// TIA Portal V16 export
// export: Created 2022-01-12T14:34:28.4377985Z, ExportSetting WithDefaults, DisplayName Totally Integrated Automation Portal, DisplayVersion V16 Update 4, DisplayName TIA Portal Version Control Interface, DisplayVersion V16 Update 2, DisplayName TIA Portal Openness, DisplayVersion V16 Update 4, DisplayName STEP 7 Professional, DisplayVersion V16 Update 4, DisplayName STEP 7 Safety, DisplayVersion V16, DisplayName WinCC Professional, DisplayVersion V16 Update 4
TYPE "typSygnałyzMaszyn"
// stored: IsFailsafeCompliant false
   STRUCT
      "M" : Array[1..5] of "typSygnały";   // maszyna
   END_STRUCT;
END_TYPE
